// TIA Portal project "2 Yönlü Motor Uygulaması" (V18)

(* hardware
DEVICE "S7-1200 station_1"  S7-1200 Station
   slot 0: "Rack_0"  S7-1200 Rack  Rack  V1.0
   slot 1: "PLC_1"  CPU 1214C AC/DC/Rly  6ES7 214-1BG40-0XB0  V4.6
*)

// ===== PLC "PLC_1"  CPU 1214C AC/DC/Rly =====

VAR_GLOBAL   // PLC tag table "Default tag table"
   "Stop" AT %I0.0 : Bool;
   "Start_1" AT %I0.1 : Bool;
   "Start_2" AT %I0.2 : Bool;
   "Motor_1" AT %Q0.0 : Bool;
   "Start_3" AT %I0.3 : Bool;
   "Saat Yönünde" AT %Q0.1 : Bool;
   "Saatin Tersi Yönde" AT %Q0.2 : Bool;
   "Aşırı Akım Koruma" AT %I0.7 : Bool;
END_VAR

ORGANIZATION_BLOCK "Main"   // OB1, LAD, ProgramCycle
TITLE = "Main Program Sweep (Cycle)"
{ S7_Optimized_Access := 'TRUE' }
VERSION : 0.1
   VAR_INPUT
      Initial_Call : Bool;   // Initial call of this OB
      Remanence : Bool;   // =True, if remanent data are available
   END_VAR
   VAR_TEMP   // added for the SCL form of the ladder/FBD networks
      _w1 : Bool;
   END_VAR
BEGIN

REGION Network 1
   // Motor iki start butonu ile iki ayrı yönde çalıştırılacaktır. 
   // Her buton bir yönde çalışma içindir. 
   // Emniyet olarak kontak emniyeti kullanılacaktır. 
   // Stop butonu ile motorun durması sağlanacaktır. 
   // Motor aşırı akım çektiğinde motorun enerjisi kesilecektir.
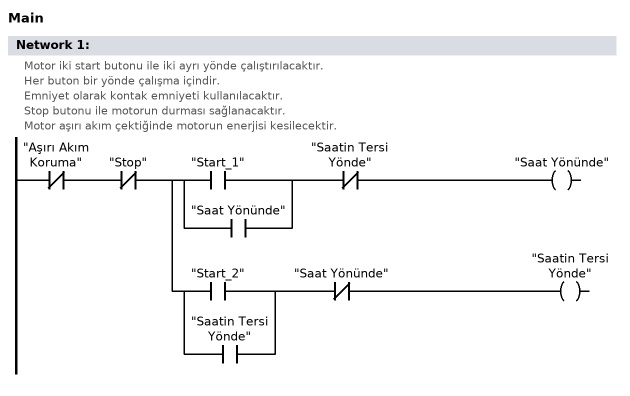
   RUNG wire#powerrail
      I_Contact( "Aşırı Akım Koruma" )
      I_Contact( "Stop" )
      wire#w1
      Contact( "Start_1" )
      wire#w2
      I_Contact( "Saatin Tersi Yönde" )
      Coil( "Saat Yönünde" )
   END_RUNG
   RUNG wire#w1
      Contact( "Saat Yönünde" )
   END_RUNG wire#w2
   RUNG wire#w1
      Contact( "Start_2" )
      wire#w3
      I_Contact( "Saat Yönünde" )
      Coil( "Saatin Tersi Yönde" )
   END_RUNG
   RUNG wire#w1
      Contact( "Saatin Tersi Yönde" )
   END_RUNG wire#w3
   // the same network as SCL:
   #_w1 := NOT "Aşırı Akım Koruma" AND NOT "Stop";
   "Saat Yönünde" := #_w1 AND ("Start_1" OR "Saat Yönünde") AND NOT "Saatin Tersi Yönde";
   "Saatin Tersi Yönde" := #_w1 AND ("Start_2" OR "Saatin Tersi Yönde") AND NOT "Saat Yönünde";
END_REGION
END_ORGANIZATION_BLOCK